{attribute 'GeneratedUsingTerminal: KL1501'}
{attribute addProperty BoxType "KL1501"}
{attribute addProperty Id "StateAT %I*USINT0Data_InAT %I*ARRAY [0..1] OF UINT0CtrlAT %Q*USINT0Data_OutAT %Q*ARRAY [0..1] OF UINT0"}
{attribute addProperty CRC "1008362752"}
{attribute addProperty Size "0"}
TYPE Channel_3C1A6500 :
STRUCT
	{attribute addProperty Name "State"}
	State AT %I* : USINT;
	{attribute addProperty Name "Data_In"}
	Data_In AT %I* : ARRAY [0..1] OF UINT;
	{attribute addProperty Name "Ctrl"}
	Ctrl AT %Q* : USINT;
	{attribute addProperty Name "Data_Out"}
	Data_Out AT %Q* : ARRAY [0..1] OF UINT;
END_STRUCT
END_TYPE

(* stored: Version 1.2.0.0, ProductVersion 3.1.4024.9
   DUT Channel_3C1A6500: Id {769c7fce-98de-444d-82b1-f8f3cfd6fc97} *)
